// TIA Portal project "SeriePareleloSetReset" (V14)

(* hardware
DEVICE "S7-1200 station_1"  S7-1200 Station
   slot 0: "Rack_0"  S7-1200 Rack  Rack  V1.0
   slot 1: "PLC_1_Testes"  CPU 1214C DC/DC/DC  6ES7 214-1AG40-0XB0  V4.2
*)

// ===== PLC "PLC_1_Testes"  CPU 1214C DC/DC/DC =====

VAR_GLOBAL   // PLC tag table "Default tag table"
   "System_Byte" AT %MB1 : Byte;
   "FirstScan" AT %M1.0 : Bool;
   "DiagStatusUpdate" AT %M1.1 : Bool;
   "AlwaysTRUE" AT %M1.2 : Bool;
   "AlwaysFALSE" AT %M1.3 : Bool;
   "Clock_Byte" AT %MB0 : Byte;
   "Clock_10Hz" AT %M0.0 : Bool;
   "Clock_5Hz" AT %M0.1 : Bool;
   "Clock_2.5Hz" AT %M0.2 : Bool;
   "Clock_2Hz" AT %M0.3 : Bool;
   "Clock_1.25Hz" AT %M0.4 : Bool;
   "Clock_1Hz" AT %M0.5 : Bool;
   "Clock_0.625Hz" AT %M0.6 : Bool;
   "Clock_0.5Hz" AT %M0.7 : Bool;
   "Tag_1" AT %M100.1 : Bool;
   "Tag_2" AT %M100.2 : Bool;
   "Tag_3" AT %Q100.1 : Bool;
   "Tag_4" AT %M100.3 : Bool;
   "Tag_5" AT %M100.4 : Bool;
   "Tag_6" AT %M100.6 : Bool;
   "Tag_7" AT %M100.7 : Bool;
END_VAR

FUNCTION "SetReset" : Void   // FC1, LAD
{ S7_Optimized_Access := 'TRUE' }
VERSION : 0.1
BEGIN

REGION Network 1: SERIE PARALELO
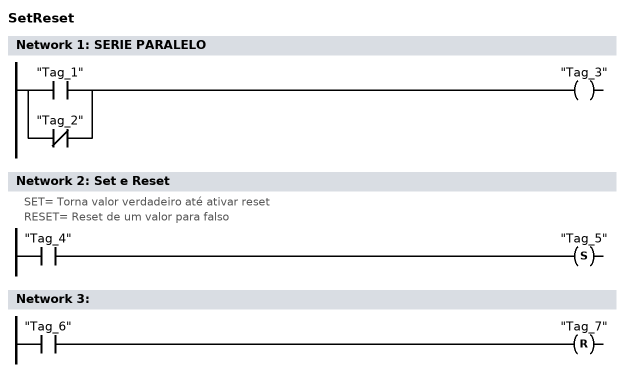
   RUNG wire#powerrail
      Contact( "Tag_1" )
      wire#w1
      Coil( "Tag_3" )
   END_RUNG
   RUNG wire#powerrail
      I_Contact( "Tag_2" )
   END_RUNG wire#w1
   // the same network as SCL:
   "Tag_3" := "Tag_1" OR NOT "Tag_2";
END_REGION

REGION Network 2: Set e Reset
   // SET= Torna valor verdadeiro até ativar reset
   // RESET= Reset de um valor para falso
   RUNG wire#powerrail
      Contact( "Tag_4" )
      S_Coil( "Tag_5" )
   END_RUNG
   // the same network as SCL:
   IF "Tag_4" THEN "Tag_5" := TRUE; END_IF;
END_REGION

REGION Network 3
   RUNG wire#powerrail
      Contact( "Tag_6" )
      R_Coil( "Tag_7" )
   END_RUNG
   // the same network as SCL:
   IF "Tag_6" THEN "Tag_7" := FALSE; END_IF;
END_REGION
END_FUNCTION

ORGANIZATION_BLOCK "Main"   // OB1, LAD, ProgramCycle
TITLE = "Main Program Sweep (Cycle)"
{ S7_Optimized_Access := 'TRUE' }
VERSION : 0.1
   VAR_INPUT
      Initial_Call : Bool;   // Initial call of this OB
      Remanence : Bool;   // =True, if remanent data are available
   END_VAR
BEGIN

REGION Network 1
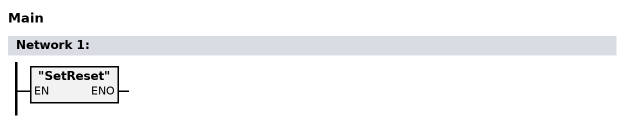
   RUNG wire#powerrail
      "SetReset"()
   END_RUNG
   // the same network as SCL:
   "SetReset"();
END_REGION
END_ORGANIZATION_BLOCK